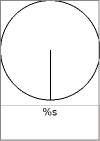
VISUALIZATION V_RotaryAxis  // 100x141
VAR_IN_OUT
	Axis : ST_AxisBase_HMI;
	Component : ST_ComponentBase_HMI;
END_VAR
    Ellipse (0,0 100x100)
    Line (50,50) (50,100)
        p2858320360: Axis.Status.ActualPositionModulo
    Textfield (0,105 100x36), "%s", text variable: Component.Config.Name
END_VISUALIZATION

(* stored: Version 1.1.0.1, ProductVersion 3.1.4024.12
   Visu V_RotaryAxis: Id {ec15b1cb-1add-4e24-8919-89e4236a57b8} *)
